(* IEC 61131-3 sources: MotionTestBenchMaster/Logical/00_AID/Libraries/Sidel_Libraries/SidelLog, 6 files *)

(* ---- SidelLog.typ ---- *)
(********************************************************************
 * COPYRIGHT --
 ********************************************************************
 * Library: SidelLog
 * File: SidelLog.typ
 * Author: Administrator
 * Created: July 15, 2014
 ********************************************************************
 * Data types of library SidelLog
 ********************************************************************)
(********************************                                    UPS LOG                                    **************************************************************)

TYPE
	Sidel_UpsIo_typ : 	STRUCT
		batteryAlarm : BOOL; (*True when the battery is failed*)
		batteryLow : BOOL; (*True when the battery is low*)
		shutdownReq : BOOL; (*Shutdown request*)
		noPowerSupply : BOOL; (*True when there is power supply*)
		shutdownAlarm : BOOL; (*True when the shutdown time exceed limits*)
		powerOffTime : UINT; (*Power off time*)
	END_STRUCT;
END_TYPE

(********************************                             SOFTWARE OBJECT LOG                **************************************************************)

TYPE
	MO_List_Light_typ : 	STRUCT
		name : ARRAY[0..13]OF SINT;
		grp : USINT;
		type : USINT;
		state : USINT;
		reserve : USINT;
		memtype : UDINT;
	END_STRUCT;
	SW_Obj_List : 	STRUCT
		version : MoVerStruc_typ; (*Version*)
		module : MO_List_Light_typ; (*Module details*)
	END_STRUCT;
END_TYPE

(* ---- LogSupplyEvents.st ---- *)
(********************************************************************
 * COPYRIGHT -- Bernecker + Rainer
 ********************************************************************
 * Library: GenUps
 * File: LogSupplyEvents.st
 * Author: gibertinim
 * Created: March 13, 2014
 ********************************************************************
 * Implementation of library GenUps
 ********************************************************************)

(* Write the power supply events in the specified logger *)
FUNCTION_BLOCK LogSupplyEvents

	IF (enable = TRUE) THEN

		CASE step OF

			0:
				pUpsIO ACCESS (ADR_UpsIO);

				errorID 			:=	ERR_FUB_BUSY;
				busy				:=	TRUE;
				error				:=	FALSE;
				noSupply			:= TRUE;
				batteryLow			:= FALSE;
				batteryAlarm		:= FALSE;
				shutdownRequested	:= FALSE;

				IF (customLogEntry_0.errorID = ERR_FUB_ENABLE_FALSE) THEN
					(* The function block started running *)
					step := 1;
				END_IF;

			1:

				memset(ADR(data),0,SIZEOF(data));
				customLogEntry_0.adrCustomEntry	:=	ADR(data);
				memset(ADR(tempString),0,SIZEOF(tempString));
				memset(ADR(tempString2),0,SIZEOF(tempString2));

				IF (pUpsIO.shutdownAlarm = TRUE) THEN
					step := 50;
				ELSE
					step := 51;
				END_IF;

			2:
				(* Waiting for an event *)

				IF 		((pUpsIO.batteryAlarm	= TRUE)		AND	(batteryAlarm		= FALSE))	THEN
					step := 10;
				ELSIF	((pUpsIO.batteryAlarm	= FALSE)	AND	(batteryAlarm		= TRUE))	THEN
					step := 11;
				ELSIF	((pUpsIO.batteryLow		= TRUE)		AND	(batteryLow			= FALSE))	THEN
					step := 20;
				ELSIF	((pUpsIO.batteryLow		= FALSE)	AND	(batteryLow			= TRUE))	THEN
					step := 21;
				ELSIF	((pUpsIO.noPowerSupply	= TRUE)		AND (noSupply			= FALSE))	THEN
					step := 30;
				ELSIF	((pUpsIO.noPowerSupply	= FALSE)	AND (noSupply			= TRUE))	THEN
					step := 31;
				ELSIF (pUpsIO.shutdownReq		= TRUE)		AND	(shutdownRequested	= FALSE)	THEN
					step := 40;
				ELSIF(	(pUpsIO.batteryAlarm	= FALSE)	AND	(batteryAlarm		= FALSE)	AND
						(pUpsIO.batteryLow		= FALSE)	AND	(batteryLow			= FALSE)	AND
						(pUpsIO.noPowerSupply	= FALSE)	AND (noSupply			= FALSE)	AND
						(pUpsIO.shutdownReq 	= FALSE)	AND (shutdownRequested	= FALSE))	THEN
					upsStatus := ERR_OK;
				ELSIF (	(pUpsIO.shutdownReq 	= FALSE)	AND (shutdownRequested	= TRUE)) THEN
					shutdownRequested := FALSE;
				END_IF;

			10:

				customLogEntry_0.enable 		:= 	TRUE;

				data.errorNum		:= ERR_UPS_BATTERY_FAULT;
				data.adr_string		:= ADR('UPS BATTERY FAULT');
				data.logLevel		:= arEVENTLOG_SEVERITY_WARNING;
				batteryAlarm		:= TRUE;
				upsStatus			:= ERR_UPS_BATTERY_FAULT;
				(* Waiting until the log is written succesfully *)
				IF (customLogEntry_0.errorID = ERR_OK) THEN
					(* Log entry written succesfully*)
					step 					:= 101;
					customLogEntry_0.enable := 	FALSE;
				ELSIF ((customLogEntry_0.errorID <> ERR_FUB_BUSY) AND (customLogEntry_0.errorID <> ERR_OK)AND (customLogEntry_0.errorID <> ERR_FUB_ENABLE_FALSE)) THEN
					(* Error occured while saving the logger *)
					errorStep	:= 10;
					errorID		:= customLogEntry_0.errorID;
					error		:= TRUE;
					step		:= 200;
				END_IF;

			11:
				(* Battery alarm recovered *)

				customLogEntry_0.enable := 	TRUE;
				data.errorNum			:= ERR_UPS_BATTERY_OK;

				data.adr_string	:= ADR('UPS BATTERY FAULT RECOVERED');
				data.logLevel	:= arEVENTLOG_SEVERITY_INFO;
				batteryAlarm	:= FALSE;
				(* Waiting until the log is written succesfully *)

				IF (customLogEntry_0.errorID = ERR_OK) THEN
					(* Log entry written succesfully*)
					step 					:= 101;
					customLogEntry_0.enable := FALSE;
				ELSIF ((customLogEntry_0.errorID <> ERR_FUB_BUSY) AND customLogEntry_0.errorID <> ERR_OK)AND (customLogEntry_0.errorID <> ERR_FUB_ENABLE_FALSE) THEN
					(* Error occured while saving the logger *)
					errorStep	:= 11;
					errorID		:= customLogEntry_0.errorID;
					error		:= TRUE;
					step		:= 200;
				END_IF;

			20:

				(* Battery low *)

				customLogEntry_0.enable 		:= 	TRUE;
				data.errorNum		:= ERR_UPS_BATTERY_LOW;
				data.adr_string		:= ADR('UPS BATTERY LOW');
				data.logLevel		:= arEVENTLOG_SEVERITY_WARNING;
				batteryLow			:= TRUE;
				upsStatus			:= ERR_UPS_BATTERY_LOW;
				(* Waiting until the log is written succesfully *)
				IF (customLogEntry_0.errorID = ERR_OK) THEN
					(* Log entry written succesfully*)
					step 					:= 101;
					customLogEntry_0.enable := FALSE;
				ELSIF ((customLogEntry_0.errorID <> ERR_FUB_BUSY) AND (customLogEntry_0.errorID <> ERR_OK)AND (customLogEntry_0.errorID <> ERR_FUB_ENABLE_FALSE)) THEN
					(* Error occured while saving the logger *)
					errorStep	:= 20;
					errorID		:= customLogEntry_0.errorID;
					error		:= TRUE;
					step		:= 200;
				END_IF;

			21:
				(* Battery recharged *)

				customLogEntry_0.enable 		:= 	TRUE;

				data.errorNum		:= ERR_UPS_BATTERY_CHARGED;
				data.adr_string		:= ADR('UPS BATTERY CHARGED');
				data.logLevel		:= arEVENTLOG_SEVERITY_INFO;
				batteryLow			:= FALSE;
				(* Waiting until the log is written succesfully *)

				IF (customLogEntry_0.errorID = ERR_OK) THEN
					(* Log entry written succesfully*)
					step 					:= 2;
					customLogEntry_0.enable := FALSE;
				ELSIF ((customLogEntry_0.errorID <> ERR_FUB_BUSY) AND (customLogEntry_0.errorID <> ERR_OK)AND (customLogEntry_0.errorID <> ERR_FUB_ENABLE_FALSE)) THEN
					(* Error occured while saving the logger *)
					errorStep	:= 21;
					errorID		:= customLogEntry_0.errorID;
					error		:= TRUE;
					step		:= 200;
				END_IF;

			30:

				(* Lost Power supply *)

				data.errorNum			:= ERR_UPS_NO_SUPPLY;
				data.adr_string			:= ADR('UPS NO POWER SUPPLY');
				data.logLevel			:= arEVENTLOG_SEVERITY_WARNING;
				noSupply				:= TRUE;
				upsStatus				:= ERR_UPS_NO_SUPPLY;
				customLogEntry_0.enable := 	TRUE;
				(* Waiting until the log is written succesfully *)
				IF (customLogEntry_0.errorID = ERR_OK) THEN
					(* Log entry written succesfully*)
					step 					:= 101;
					customLogEntry_0.enable := FALSE;
				ELSIF ((customLogEntry_0.errorID<> ERR_FUB_BUSY) AND (customLogEntry_0.errorID <> ERR_OK)AND (customLogEntry_0.errorID <> ERR_FUB_ENABLE_FALSE)) THEN
					(* Error occured while saving the logger *)
					errorStep	:= 30;
					errorID		:= customLogEntry_0.errorID;
					error		:= TRUE;
					step		:= 200;
				END_IF;

			31:
				(* Power supply ok *)

				customLogEntry_0.enable 		:= 	TRUE;

				data.errorNum		:= ERR_UPS_SUPPLY_BACK;
				data.adr_string		:= ADR('UPS POWER SUPPLY OK');
				data.logLevel		:= arEVENTLOG_SEVERITY_INFO;
				noSupply			:= FALSE;
				(* Waiting until the log is written succesfully *)
				IF (customLogEntry_0.errorID = ERR_OK) THEN
					(* Log entry written succesfully*)
					step 					:= 101;
					customLogEntry_0.enable := FALSE;
				ELSIF ((customLogEntry_0.errorID <> ERR_FUB_BUSY) AND (customLogEntry_0.errorID <> ERR_OK) AND (customLogEntry_0.errorID <> ERR_FUB_ENABLE_FALSE)) THEN
					(* Error occured while saving the logger *)
					errorStep	:= 31;
					errorID		:= customLogEntry_0.errorID;
					error		:= TRUE;
					step		:= 200;
				END_IF;

			40:
				(* Shutdown request *)

				customLogEntry_0.enable 		:= 	TRUE;

				data.errorNum		:= ERR_UPS_SHUTDOWN_REQ;
				data.adr_string		:= ADR('UPS SHUTDOWN REQUEST');
				data.logLevel		:= arEVENTLOG_SEVERITY_INFO;
				shutdownRequested	:= TRUE;
				upsStatus			:= ERR_UPS_SHUTDOWN_REQ;
				(* Waiting until the log is written succesfully *)
				IF (customLogEntry_0.errorID = ERR_OK) THEN
					(* Log entry written succesfully*)
					step 					:= 101;
					customLogEntry_0.enable := FALSE;
				ELSIF ((customLogEntry_0.errorID <> ERR_FUB_BUSY) AND (customLogEntry_0.errorID <> ERR_OK) AND (customLogEntry_0.errorID <> ERR_FUB_ENABLE_FALSE)) THEN
					(* Error occured while saving the logger *)
					errorStep	:= 40;
					errorID		:= customLogEntry_0.errorID;
					error		:= TRUE;
					step		:= 200;
				END_IF;

			50:
				(* Writing the total power off time to the logger *)
				(* Shutdown request *)
				itoa(pUpsIO.powerOffTime, ADR(tempString));
				tempString2 := 'UPS SHUTDOWN TIME ';
				strcat(ADR(tempString2), ADR(tempString));
				strcat(ADR(tempString2), ADR('s'));

				customLogEntry_0.enable 		:= 	TRUE;
				data.errorNum					:= ERR_UPS_SHUTDOWN_TIME;
				data.adr_string					:= ADR(tempString2);
				data.logLevel					:= arEVENTLOG_SEVERITY_INFO;
				shutdownRequested				:= TRUE;
				upsStatus						:= ERR_UPS_SHUTDOWN_REQ;

				(* Waiting until the log is written succesfully *)
				IF (customLogEntry_0.errorID = ERR_OK) THEN
					(* Log entry written succesfully*)
					step 					:= 51;
					customLogEntry_0.enable := FALSE;
				ELSIF ((customLogEntry_0.errorID <> ERR_FUB_BUSY) AND (customLogEntry_0.errorID <> ERR_OK) AND (customLogEntry_0.errorID <> ERR_FUB_ENABLE_FALSE)) THEN
					(* Error occured while saving the logger *)
					errorStep	:= 50;
					errorID		:= customLogEntry_0.errorID;
					error		:= TRUE;
					step		:= 200;
				END_IF;

			51:

				(* Identifier obtained succesfully *)
				IF (pUpsIO.noPowerSupply = TRUE) THEN
					step := 30;
				ELSE
					step := 31;
				END_IF;

			100:
				(* Waiting until the log is written succesfully *)
				IF (customLogEntry_0.errorID = ERR_OK) THEN
					(* Log entry written succesfully*)
					step := 101;

				ELSIF ((customLogEntry_0.errorID <> ERR_FUB_BUSY) AND (customLogEntry_0.errorID <> ERR_OK) AND (customLogEntry_0.errorID <> ERR_FUB_ENABLE_FALSE)) THEN
					(* Error occured while saving the logger *)
					errorStep	:= 100;
					errorID		:= customLogEntry_0.errorID;
					error		:= TRUE;
					step		:= 200;
				END_IF

			101:
			(* Disabling the function block *)
				IF (customLogEntry_0.errorID = ERR_FUB_ENABLE_FALSE) THEN
					memset(ADR(data),0,SIZEOF(data));
					step 			:= 2;
				END_IF;

			200:
			(* Error step *)
				customLogEntry_0.enable	:=	FALSE;

		END_CASE;

	ELSE

		error					:= TRUE;
		errorID					:= ERR_FUB_ENABLE_FALSE;
		customLogEntry_0.enable	:=	FALSE;
		step					:= 0;
		errorStep				:= 0;
		upsStatus				:= ERR_OK;
		noSupply				:= TRUE;
		batteryLow				:= FALSE;
		batteryAlarm			:= FALSE;
		shutdownRequested		:= FALSE;
		busy					:= FALSE;
		memset(ADR(data),0,SIZEOF(data));
	END_IF;

	customLogEntry_0();
END_FUNCTION_BLOCK

(* ---- SidelLog.fun ---- *)
(********************************************************************
 * COPYRIGHT --
 ********************************************************************
 * Library: SidelLog
 * File: SidelLog.fun
 * Author: Administrator
 * Created: July 15, 2014
 ********************************************************************
 * Functions and function blocks of library SidelLog
 ********************************************************************)

FUNCTION_BLOCK LogSupplyEvents (*Write the power supply events in the specified logger*)
	VAR_INPUT
		enable : BOOL; (*Enable the execution of the function block*)
		ADR_UpsIO : UDINT; (*Address of the UPS IO interface*)
	END_VAR
	VAR_OUTPUT
		errorID : DINT; (*Current error ID*)
		error : BOOL; (*True when the function block is in error*)
		upsStatus : UINT; (*Ups output status*)
		busy : BOOL; (*True when the function block is running*)
		errorStep : USINT; (*Error step*)
	END_VAR
	VAR
		step : USINT; (*Internal step*)
		batteryAlarm : BOOL; (*True when the battery is in alarm*)
		batteryLow : BOOL; (*True when the battery is low*)
		shutdownRequested : BOOL; (*Shutdown requested*)
		noSupply : BOOL; (*True wjen the power supply failed*)
		pUpsIO : REFERENCE TO Sidel_UpsIo_typ; (*Pointer to the UPS IO interface*)
		customLogEntry_0 : CustomLogEntry; (*Wrinting and getting information into a specified Logger*)
		tempString2 : STRING[80];
		tempString : STRING[80];
		data : pwr_log_custom_entry; (*Internal data to write*)
	END_VAR
END_FUNCTION_BLOCK

FUNCTION_BLOCK SynchLog (*Machine synchronization logger*)
	VAR_INPUT
		enable : BOOL; (*Enable the execution of the function block*)
		RAX1 : USINT;
		AXN : USINT;
		offsetAcquire : BOOL;
		testBit : USINT;
		axisNameHoming : STRING[80];
		axisName : STRING[80];
		positionMm : REAL;
		positionMmHoming : REAL;
	END_VAR
	VAR_OUTPUT
		errorID : DINT; (*Current error ID*)
		error : BOOL; (*True when the function block is in error*)
		testIndex : USINT;
		busy : BOOL; (*True when the function block is running*)
	END_VAR
	VAR
		step : USINT; (*Internal step*)
		errorStep : USINT; (*Error step*)
		indexAxis : USINT;
		phasingString : STRING[80];
		phasingAxisPosition : STRING[80];
		data : pwr_log_custom_entry; (*Wrinting and getting information into a specified Logger*)
		customLogEntry_0 : CustomLogEntry; (*Internal data to write*)
		rTrig_0 : R_TRIG;
	END_VAR
END_FUNCTION_BLOCK

FUNCTION_BLOCK SwChg (*Monitor and write into the user logger the canges of the software objects*)
	VAR_INPUT
		enable : BOOL; (*Enable the function block*)
		logLevel : USINT; (*Level of the log entry*)
		refreshTime : TIME; (*Refresh time*)
	END_VAR
	VAR_OUTPUT
		scan : BOOL; (*True when the module is getting the software object list*)
		searching : BOOL; (*True when the function block is searching for software object changes*)
		writingLog : BOOL; (*True when the funciton block is writing the entry into the logger*)
		waiting : BOOL; (*Waiting to search again*)
		busy : BOOL; (*True when the function block is busy*)
		error : BOOL; (*True when the function block is in error*)
		errorID : DINT; (*Actual error ID*)
	END_VAR
	VAR
		errorSubStep : USINT; (*Internal error SubStep*)
		errorStep : USINT; (*Internal erro Step*)
		step : USINT; (*Internal step*)
		substep : USINT; (*Internal substep*)
		cnt : UDINT; (*Internal counter*)
		mo_prev_index : UINT; (*List previous index*)
		mo_index : UINT; (*Actual index*)
		refresh : TON; (*Refresh timer*)
		waitWrite : TON; (*CF data object write delay*)
		customEntry : pwr_log_custom_entry; (*Custom log entry*)
		tempString : STRING[80]; (*Temporary string*)
		tempModule : MO_List_typ; (*Temporary module informations*)
		nrChanges : UINT; (*Number of changed elements*)
		swListTempID : UDINT; (*Temporary software list ID*)
		swListID : UDINT; (*Software list ID*)
		iOldList : ARRAY[0..iMaxEntries] OF SW_Obj_List; (*Internal Old List*)
		iActList : ARRAY[0..iMaxEntries] OF SW_Obj_List; (*Internal Actual List*)
	END_VAR
	VAR CONSTANT
		CST_fwOBJ : USINT := 132; (*Firmware Object*)
		CST_configOBJ : USINT := 67; (*Configuration Object*)
		CST_hwOBJ : USINT := 43; (*Hrdwa object*)
		CST_ncOBJ : USINT := 70; (*NC Object*)
		CST_cycOBJ : USINT := 17; (*Cyclic Object*)
		CST_sysOBJ : USINT := 18; (*System Object*)
		iMaxEntries : UINT := 999; (*Internal number of entries*)
	END_VAR
	VAR
		writeDiff : CustomLogEntry; (*Writes the custom information into the logger*)
		datObjWrite_0 : DatObjWrite; (*Write into a data Object*)
		datObjRead_0 : DatObjRead; (*Read data from a data Object*)
		datObjInfo_0 : DatObjInfo; (*Get the informations from a data object*)
		datObjCopy_0 : DatObjCopy; (*Copy a data object*)
		datObjCreate_0 : DatObjCreate; (*Create a data object*)
		datObjDelete_0 : DatObjDelete; (*Delete a data object*)
		actListElements : UINT; (*Number of entries in the actual list*)
		oldListElements : UINT; (*Number of entries in the old list*)
		newSwListT : BOOL; (*Software list data object present*)
		oldSubStep : USINT;
	END_VAR
END_FUNCTION_BLOCK

(* ---- SwChg.st ---- *)
(********************************************************************
 * COPYRIGHT --
 ********************************************************************
 * Library: Powertoys
 * File: swChg.st
 * Author: Massimo Gibertini
 * Created: August 07, 2014
 ********************************************************************
 * Implementation of library Powertoys
 ********************************************************************)

(* Monitor and write into the user logger the canges of the software objects *)
FUNCTION_BLOCK SwChg

	IF (enable = TRUE) THEN
		customEntry.logLevel 		:= logLevel;
		waitWrite.PT				:= T#10m;

		CASE step OF

			0:
				(* Getting the software list *)
				busy			:= TRUE;
				searching		:= FALSE;
				writingLog		:= FALSE;
				waiting			:= FALSE;
				scan			:= TRUE;
				error			:= FALSE;
				errorID			:= ERR_FUB_BUSY;

				CASE substep OF

					0:
						memset(ADR(tempModule),0,SIZEOF(tempModule));
						memset(ADR(iActList),0,SIZEOF(iActList));
						memset(ADR(iOldList),0,SIZEOF(iOldList));

						(* Checking if the swList temporary data object exist in the userRam or not*)
						datObjInfo_0.pName 	:= ADR(swListTempDataObjName);
						datObjInfo_0.enable	:= TRUE;
						substep 			:= 1;

					1:
						datObjInfo_0();
						IF (datObjInfo_0.status = doERR_MODULNOTFOUND) THEN
							(* Temporary data object not found *)
							swListTempID	:= 0;
							substep			:= 5;
						ELSIF (datObjInfo_0.status = ERR_OK) THEN
							(* Data object found *)
							swListTempID	:= datObjInfo_0.ident;
							//substep			:= 2;
							substep			:= 5;
						ELSIF (datObjInfo_0.status <> ERR_OK) AND (datObjInfo_0.status <> doERR_MODULNOTFOUND) AND (datObjInfo_0.status <> ERR_FUB_BUSY) THEN
							errorID			:= datObjInfo_0.status;
							errorStep		:= step;
							errorSubStep	:= substep;
							step 			:= 200;
							substep			:= 0;
						END_IF;

					2:
						datObjInfo_0.enable	:= FALSE;
						datObjInfo_0();
						IF (datObjInfo_0.status = ERR_FUB_ENABLE_FALSE) THEN
							substep			:= 3;
						END_IF;

					3:
						(* Delete the temporary data object *)
						datObjDelete_0.ident	:= swListTempID;
						datObjDelete_0.enable	:= TRUE;
						substep					:= 4;

					4:
						datObjDelete_0();
						IF (datObjDelete_0.status = ERR_OK) THEN
							substep			:= 5;
							swListTempID	:= 0;
						ELSIF (datObjDelete_0.status <> ERR_OK) AND (datObjDelete_0.status <> ERR_FUB_BUSY) THEN
							errorID			:= datObjDelete_0.status;
							errorStep		:= step;
							errorSubStep	:= substep;
							step 			:= 200;
							substep			:= 0;
						END_IF;

					5:
						(* Disable fub *)
						datObjDelete_0.enable	:= FALSE;
						datObjDelete_0();
						datObjInfo_0.enable	:= FALSE;
						datObjInfo_0();
						IF (datObjDelete_0.status = ERR_FUB_ENABLE_FALSE) AND (datObjInfo_0.status = ERR_FUB_ENABLE_FALSE) THEN
							substep				:= 6;
						END_IF;

					6:
						(* temporary data object not present or deleted *)
						(* Checking if the swList data object exist or not *)
						datObjInfo_0.pName 	:= ADR(swListDatObjName);
						datObjInfo_0.enable	:= TRUE;
						datObjInfo_0();
						IF (datObjInfo_0.status <> ERR_FUB_BUSY) AND (datObjInfo_0.status <> ERR_FUB_ENABLE_FALSE) THEN
							substep := 7;
						END_IF;

					7:
						datObjInfo_0();
						IF (datObjInfo_0.status = doERR_MODULNOTFOUND) THEN
							(* Data object not found *)
							swListID		:= 0;
							substep			:= 100;
						ELSIF (datObjInfo_0.status = doERR_CHECKSUM_WARNING) THEN
							swListID		:= datObjInfo_0.ident;
							substep			:= 10;
						ELSIF (datObjInfo_0.status = ERR_OK) THEN
							(* Data object found *)
							swListID		:= datObjInfo_0.ident;
							IF (swListTempID = 0) THEN
								substep			:= 50;
							ELSE
								substep 		:= 150;
							END_IF;

						ELSIF (datObjInfo_0.status <> ERR_OK) AND (datObjInfo_0.status <> doERR_CHECKSUM_WARNING) AND (datObjInfo_0.status <> doERR_MODULNOTFOUND) AND (datObjInfo_0.status <> ERR_FUB_BUSY) THEN
							errorID			:= datObjInfo_0.status;
							errorStep		:= step;
							errorSubStep	:= substep;
							step 			:= 200;
							substep			:= 0;
						END_IF;

					(* Data object damaged, deleting *)
					10:
						datObjInfo_0.enable	:= FALSE;
						datObjInfo_0();
						IF (datObjInfo_0.status = ERR_FUB_ENABLE_FALSE) THEN
							substep			:= 11;
						END_IF;

					11:
						datObjDelete_0.ident	:= swListID;
						datObjDelete_0.enable	:= TRUE;
						datObjDelete_0();
						IF (datObjDelete_0.status <> ERR_FUB_BUSY) AND (datObjDelete_0.status <> ERR_FUB_ENABLE_FALSE) THEN
							substep 				:= 12;
						END_IF;

					12:
						datObjDelete_0();
						IF (datObjDelete_0.status = ERR_OK) THEN
							substep				:= 13;
						ELSIF (datObjDelete_0.status <> ERR_OK) AND (datObjDelete_0.status <> ERR_FUB_BUSY) THEN
							errorID				:= datObjDelete_0.status;
							errorStep			:= step;
							errorSubStep		:= substep;
							step 				:= 200;
							substep				:= 0;
						END_IF;

					13:
						datObjDelete_0.enable	:= FALSE;
						datObjDelete_0();
						IF (datObjDelete_0.status = ERR_FUB_ENABLE_FALSE) THEN
							(* No existing data object *)
							substep 			:= 100;
							swListID 			:= 0;
						END_IF;

					50:
						(* swList data object present, copy to DRam *)
						datObjInfo_0.enable			:= FALSE;
						datObjCopy_0.ident 			:= swListID;
						datObjCopy_0.pNameTarget 	:= ADR(swListTempDataObjName);
						datObjCopy_0.MemTypeTarget	:= doTEMP;
						datObjCopy_0.enable			:= TRUE;
						datObjCopy_0();
						substep := 51;

					51:
						datObjCopy_0();
						IF (datObjCopy_0.status = ERR_OK) THEN
							substep 				:= 52;
							swListTempID			:= datObjCopy_0.identNew;
						ELSIF (datObjCopy_0.status <> ERR_OK) AND (datObjCopy_0.status <> ERR_FUB_BUSY) THEN
							errorID					:= datObjCopy_0.status;
							errorStep				:= step;
							errorSubStep			:= substep;
							step 					:= 200;
							substep					:= 0;
						END_IF;

					52:
						datObjCopy_0.enable			:= FALSE;
						datObjCopy_0();
						IF (datObjCopy_0.status = ERR_FUB_ENABLE_FALSE) THEN
							(* Temporary Data object recovered succesfully *)
							substep					:= 150;

						END_IF;

					100:
						(* Creating the temporary data object*)
						IF (swListTempID = 0) THEN
							datObjInfo_0.enable		:= FALSE;
							datObjCreate_0.grp		:= 0;
							datObjCreate_0.pName	:= ADR(swListTempDataObjName);
							datObjCreate_0.len		:= SIZEOF(iActList);
							datObjCreate_0.MemType	:= doTEMP;
							datObjCreate_0.Option	:= doNO_CS;
							datObjCreate_0.pCpyData	:= ADR(iActList);
							datObjCreate_0.enable	:= TRUE;
							datObjCreate_0();
							substep					:= 101;
						ELSE
							substep					:= 110;
						END_IF;

					101:
						datObjCreate_0();
						IF (datObjCreate_0.status = ERR_OK) THEN
							substep				:= 102;
							swListTempID		:= datObjCreate_0.ident;
							newSwListT			:= TRUE;
						ELSIF (datObjCreate_0.status <> ERR_OK) AND (datObjCreate_0.status <> ERR_FUB_BUSY) THEN
							errorID				:= datObjCreate_0.status;
							errorStep			:= step;
							errorSubStep		:= substep;
							step 				:= 200;
							substep				:= 0;
						END_IF;

					102:
						datObjCreate_0.enable	:= FALSE;
						datObjCreate_0();
						IF (datObjCreate_0.status = ERR_FUB_ENABLE_FALSE) THEN
							substep				:= 110;

						END_IF;

					110:
						(* Creating the cf data object*)
						datObjCreate_0.grp		:= 0;
						datObjCreate_0.pName	:= ADR(swListDatObjName);
						datObjCreate_0.len		:= SIZEOF(iOldList);
						datObjCreate_0.MemType	:= doUSRROM;
						datObjCreate_0.Option	:= 0;
						datObjCreate_0.pCpyData	:= ADR(iOldList);
						datObjCreate_0.enable	:= TRUE;
						substep					:= 112;

					112:
						datObjCreate_0();
						IF (datObjCreate_0.status = ERR_OK) THEN
							substep					:= 113;
							swListID				:= datObjCreate_0.ident;
							datObjCreate_0.enable	:= FALSE;
						ELSIF (datObjCreate_0.status <> ERR_OK) AND (datObjCreate_0.status <> ERR_FUB_BUSY) THEN
							errorID					:= datObjCreate_0.status;
							errorStep				:= step;
							errorSubStep			:= substep;
							step 					:= 200;
							substep					:= 0;
						END_IF;

					113:
						datObjCreate_0.enable		:= FALSE;
						datObjCreate_0();
						IF (datObjCreate_0.status = ERR_FUB_ENABLE_FALSE) AND newSwListT THEN
							substep					:= 200;
							oldListElements			:= 0;
						ELSIF (datObjCreate_0.status = ERR_FUB_ENABLE_FALSE) AND NOT (newSwListT) THEN
							substep					:= 150;
							oldListElements			:= 0;
						END_IF;

					150:
						(* Loading the existing temporary data object *)
						datObjRead_0.ident			:= swListTempID;
						datObjRead_0.Offset			:= 0;
						datObjRead_0.pDestination	:= ADR(iOldList);
						datObjRead_0.len			:= SIZEOF(iOldList);
						datObjRead_0.enable			:= TRUE;
						datObjRead_0();
						substep						:= 151;

					151:

						datObjRead_0();
						IF (datObjRead_0.status = ERR_OK) THEN
							substep					:= 152;
						ELSIF (datObjRead_0.status <> ERR_OK) AND (datObjRead_0.status <> ERR_FUB_BUSY)	THEN
							errorID					:= datObjRead_0.status;
							errorStep				:= step;
							errorSubStep			:= substep;
							step 					:= 200;
							substep					:= 0;
						END_IF;

					152:
						datObjRead_0.enable			:= FALSE;
						datObjRead_0();
						IF (datObjRead_0.status = ERR_FUB_ENABLE_FALSE) THEN
							oldListElements 		:= 0;
							substep 				:= 153;
						END_IF;

					153:
						(* Listing the number of entries in the old list *)
						memset(ADR(tempString),0,SIZEOF(tempString));
						memcpy(ADR(tempString),ADR(iOldList[oldListElements].module.name[0]),SIZEOF(iOldList[oldListElements].module.name));
						IF (tempString <> '') THEN
							oldListElements := oldListElements + 1;
						ELSE
							substep 		:= 200;
						END_IF;

					200:
						(* Cleaning the memory of the actual list *)
						(* Listing all the software objects *)
						memset(ADR(iActList),0,SIZEOF(iActList));
						mo_prev_index 	:= 16#FFFF;
						mo_index 		:= 0;
						nrChanges 		:= 0;
						substep			:= 201;

					201:
						(* Listing all the software objects element *)
						memset(ADR(tempModule), 0, SIZEOF(tempModule));
						MO_list(mo_prev_index, ADR(mo_index),ADR(tempModule));

						IF (tempModule.type <> 0) AND ((tempModule.type = CST_configOBJ)	OR
							(tempModule.type = CST_cycOBJ)		OR
							(tempModule.type = CST_fwOBJ)		OR
							(tempModule.type = CST_hwOBJ)		OR
							(tempModule.type = CST_ncOBJ)		OR
							(tempModule.type = CST_sysOBJ))		THEN

							(* Valid system object *)
							MO_ver(ADR(tempModule.name),0,ADR(iActList[nrChanges].version));
							memcpy(ADR(iActList[nrChanges].module.name[0]),ADR(tempModule.name[0]), SIZEOF(tempModule.name));

							iActList[nrChanges].module.grp		:= tempModule.grp;
							iActList[nrChanges].module.memtype	:= tempModule.memtype;
							iActList[nrChanges].module.reserve 	:= tempModule.reserve;
							iActList[nrChanges].module.state	:= tempModule.state;
							iActList[nrChanges].module.type		:= tempModule.type;

							nrChanges							:= nrChanges + 1;
							substep 							:= 202;
						ELSE
							substep 							:= 202;
						END_IF;

					202:
						(* Checking if I have finished to scan *)

						IF (mo_prev_index = mo_index) OR (nrChanges = iMaxEntries) THEN
							substep 		:= 203;
						ELSE
							mo_prev_index	:= mo_index;
							substep 		:= 201;
						END_IF;

					203:
						(* Software list complete *)
						actListElements 	:= nrChanges;
						step 				:= 1;
						substep 			:= 0;

				END_CASE;

			1:
				(* Searching for modified software objects *)
				busy			:= TRUE;
				searching		:= TRUE;
				writingLog		:= FALSE;
				waiting			:= FALSE;
				scan			:= FALSE;
				error			:= FALSE;
				errorID			:= ERR_FUB_BUSY;

				CASE substep OF
					0:
						(* Software list complete, comparing memory area *)
						IF (memcmp(ADR(iActList), ADR(iOldList), SIZEOF(iActList)) = 0) THEN

							(* No software changes *)
							substep	:= 0;
							step	:= 20;

						ELSE

							(* There are some changes *)
							substep		:= 1;
							cnt			:= 0;
							nrChanges	:= 0;
							oldSubStep	:= 0;
						END_IF;

					1:
						(* Trying to find the module in the same position of the old array *)
						(* First speed up improvement *)
						IF ((memcmp(ADR(iActList[nrChanges].module.name[0]), ADR(iOldList[nrChanges].module.name[0]), SIZEOF(iOldList[nrChanges].module.name)) = 0)
							AND (cnt < oldListElements) AND (nrChanges < actListElements)) THEN

							(* Module found *)
							IF (memcmp(ADR(iActList[nrChanges]),ADR(iOldList[nrChanges]),SIZEOF(iOldList[nrChanges])) = 0) THEN

								(* The module are the same *)
								nrChanges	:= nrChanges + 1;
								cnt			:= 0;
							ELSE

								(* The module is modified *)
								substep 	:= 10;
								step		:= 10;

							END_IF;

						ELSE
							(* Module not found *)
							substep 	:= 10;

						END_IF;

					10:
						(* Comparing the all elements of the iActList with all the elements of iOldList to find if the element exist or not *)
						IF (memcmp(ADR(iActList[nrChanges].module.name[0]), ADR(iOldList[cnt].module.name[0]), SIZEOF(iOldList[cnt].module.name)) <> 0) AND (nrChanges < actListElements) THEN
							IF (cnt < oldListElements)  THEN
								(* Module not found *)
								cnt 		:= cnt + 1;

							ELSIF (cnt >= oldListElements)  THEN

								(* New software module *)
								substep		:= 20;
								step		:= 10;
							END_IF;

						ELSIF ((memcmp(ADR(iActList[nrChanges].module.name[0]), ADR(iOldList[cnt].module.name[0]), SIZEOF(iOldList[cnt].module.name)) = 0)
								AND (cnt < oldListElements) AND (nrChanges < actListElements)) THEN

							(* Module found *)
							IF (memcmp(ADR(iActList[nrChanges]),ADR(iOldList[cnt]),SIZEOF(iOldList[cnt])) = 0) THEN

								(* The module are the same *)
								nrChanges	:= nrChanges + 1;
								cnt			:= 0;
								substep 	:= 1;
							ELSE

								(* The module is modified *)
								substep 	:= 10;
								step		:= 10;
							END_IF;

						ELSIF (nrChanges >= actListElements) THEN

							(* Search finished, checking the removed objects *)
							substep			:= 2;
							cnt 			:= 0;
							nrChanges 		:= 0;
						END_IF;

					2:
						(* Trying to find the module in the same position of the old array *)
						(* Second speed up improvement *)
						IF ((memcmp(ADR(iActList[cnt].module.name[0]), ADR(iOldList[cnt].module.name[0]), SIZEOF(iOldList[cnt].module.name)) = 0)
							AND (cnt < oldListElements) AND (nrChanges < actListElements)) THEN

							(* Module found *)
							cnt				:= cnt + 1;
							nrChanges		:= 0;

						ELSE
							(* Module not found *)
							nrChanges		:= 0;
							substep 	:= 20;
						END_IF

					20:
						(* Checking if there are any removed software object *)
						IF (memcmp(ADR(iActList[nrChanges].module.name[0]), ADR(iOldList[cnt].module.name[0]), SIZEOF(iOldList[cnt].module.name)) <> 0) AND (oldListElements <> 0) AND (cnt < oldListElements) THEN

							IF  (nrChanges < actListElements) THEN

								(* Module not found *)
								nrChanges	:= nrChanges + 1;

							ELSIF (nrChanges >= actListElements) THEN

								(* SW module removed *)
								substep 	:= 0;
								step		:= 10;
							END_IF;

						ELSIF ((memcmp(ADR(iActList[nrChanges].module.name[0]), ADR(iOldList[cnt].module.name[0]), SIZEOF(iOldList[cnt].module.name)) = 0)
							AND (cnt < oldListElements) AND (nrChanges < actListElements)) THEN

							(* Module found *)
							cnt				:= cnt + 1;
							substep 		:= 2;
							nrChanges		:= 0;

						ELSIF (cnt >= oldListElements) THEN

							(* Search finished *)
							step			:= 10;
							substep 		:= 30;
							cnt				:= 0;
							nrChanges		:= 0;
						END_IF;

				END_CASE;

			10:
				(* Writing informations into the logger and data object *)
				busy 			:= TRUE;
				searching 		:= FALSE;
				writingLog		:= TRUE;
				waiting 		:= FALSE;
				scan			:= FALSE;
				error			:= FALSE;
				errorID			:= ERR_FUB_BUSY;

				CASE substep OF

					0:
						(* Removed software module *)
						memset(ADR(tempString),0,SIZEOF(tempString));
						tempString	:= 'REMOVED SW MODULE: ';
						memcpy(ADR(tempString)+LEN(tempString),ADR(iOldList[cnt].module.name[0]), SIZEOF(iOldList[cnt].module.name));
						substep		:= 1;

					1:
						(* Writing into the logger *)
						customEntry.adr_string 		:= ADR(tempString);
						customEntry.errorNum 		:= LOG_SW_OBJ_CHG;
						writeDiff.adrCustomEntry 	:= ADR(customEntry);
						writeDiff.enable 			:= TRUE;
						substep 					:= 2;

					2:

						IF (writeDiff.done = TRUE) THEN
							substep			:= 3;
						ELSIF (writeDiff.error) THEN
							errorID			:= writeDiff.errorID;
							errorStep		:= step;
							errorSubStep	:= substep;
							step 			:= 200;
							substep			:= 0;
						END_IF;

					3:
						writeDiff.enable	:= FALSE;
						IF (writeDiff.errorID = ERR_FUB_ENABLE_FALSE) THEN
							cnt				:= cnt + 1;
							nrChanges		:= 0;
							step			:= 1;
							substep			:= 2;
						END_IF;

					10:
						(* Modified software module *)
						memset(ADR(tempString),0,SIZEOF(tempString));
						tempString	:= 'MODIFIED SW MODULE: ';
						memcpy(ADR(tempString)+LEN(tempString),ADR(iActList[nrChanges].module.name[0]), SIZEOF(iActList[nrChanges].module.name));
						substep		:= 11;

					11:
						(* Writing into the logger *)
						customEntry.adr_string 		:= ADR(tempString);
						customEntry.errorNum 		:= LOG_SW_OBJ_CHG;
						writeDiff.adrCustomEntry 	:= ADR(customEntry);
						writeDiff.enable 			:= TRUE;
						substep 					:= 12;

					12:

						IF (writeDiff.done = TRUE) THEN
							substep			:= 13;
						ELSIF (writeDiff.error) THEN
							errorID			:= writeDiff.errorID;
							errorStep		:= step;
							errorSubStep	:= substep;
							step 			:= 200;
							substep			:= 0;
						END_IF;

					13:
						writeDiff.enable	:= FALSE;
						IF (writeDiff.errorID = ERR_FUB_ENABLE_FALSE) THEN
							cnt				:= 0;
							nrChanges		:= nrChanges + 1;
							substep			:= 1;
							step			:= 1;
						END_IF;

					20:
						(* New software module *)
						memset(ADR(tempString),0,SIZEOF(tempString));
						tempString	:= 'NEW SW MODULE: ';
						memcpy(ADR(tempString)+LEN(tempString),ADR(iActList[nrChanges].module.name[0]), SIZEOF(iActList[nrChanges].module.name));
						substep		:= 21;

					21:
						(* Writing into the logger *)
						customEntry.adr_string 		:= ADR(tempString);
						customEntry.errorNum 		:= LOG_SW_OBJ_NEW;
						writeDiff.adrCustomEntry 	:= ADR(customEntry);
						writeDiff.enable 			:= TRUE;
						substep						:= 22;

					22:
						IF (writeDiff.done = TRUE) THEN
							substep			:= 23;
						ELSIF (writeDiff.error) THEN
							errorID			:= writeDiff.errorID;
							errorStep		:= step;
							errorSubStep	:= substep;
							step 			:= 200;
							substep			:= 0;
						END_IF;

					23:
						writeDiff.enable	:= FALSE;
						IF (writeDiff.errorID = ERR_FUB_ENABLE_FALSE) THEN
							cnt				:= 0;
							nrChanges		:= nrChanges + 1;
							substep			:= 1;
							step			:= 1;
						END_IF;

					30:
						(* Writing temporary data object *)
						datObjWrite_0.ident		:= swListTempID;
						datObjWrite_0.len		:= SIZEOF(iActList);
						datObjWrite_0.Offset	:= 0;
						datObjWrite_0.pSource	:= ADR(iActList);
						datObjWrite_0.enable	:= TRUE;
						datObjWrite_0();
						substep					:= 31;

					31:
						datObjWrite_0();
						IF (datObjWrite_0.status = ERR_OK) THEN
							substep 				:= 50;
							waitWrite.IN 			:= TRUE;
							datObjWrite_0.enable 	:= FALSE;
						ELSIF (datObjWrite_0.status <> ERR_OK) AND (datObjWrite_0.status <> ERR_FUB_BUSY) THEN
							errorID					:= datObjWrite_0.status;
							errorStep				:= step;
							errorSubStep			:= substep;
							step 					:= 200;
							substep					:= 0;
						END_IF;

					40:
						(* Writing cf data object *)
						datObjWrite_0.ident			:= swListID;
						datObjWrite_0.len			:= SIZEOF(iActList);
						datObjWrite_0.Offset		:= 0;
						datObjWrite_0.pSource		:= ADR(iActList);
						datObjWrite_0.enable		:= TRUE;
						datObjWrite_0();
						substep						:= 41;
					41:
						datObjWrite_0();
						IF (datObjWrite_0.status = ERR_OK) THEN
							substep 				:= 50;
							waitWrite.IN 			:= FALSE;
							datObjWrite_0.enable 	:= FALSE;
						ELSIF (datObjWrite_0.status <> ERR_OK) AND (datObjWrite_0.status <> ERR_FUB_BUSY) THEN
							errorID					:= datObjWrite_0.status;
							errorStep				:= step;
							errorSubStep			:= substep;
							step 					:= 200;
							substep					:= 0;
						END_IF;

					50:
						(* Copy the actual list into the old list *)
						memcpy(ADR(iOldList), ADR(iActList), SIZEOF(iActList));
						memset(ADR(tempString),0,SIZEOF(tempString));
						substep := 0;
						step 	:= 20;
				END_CASE;

			20:
				(* Waiting step *)
				busy 			:= TRUE;
				searching 		:= FALSE;
				writingLog		:= FALSE;
				waiting 		:= TRUE;
				scan			:= FALSE;
				error			:= FALSE;
				errorID			:= ERR_FUB_BUSY;

				CASE substep OF
					0:
						(* No software changes *)
						refresh.PT := refreshTime;
						refresh.IN := TRUE;

						IF refresh.Q THEN
							substep := 1;
						END_IF;

					1:
						(* Refresh time elapsed *)
						IF (waitWrite.Q) THEN
							step 	:= 10;
							substep := 40;
						ELSE
							refresh.IN := FALSE;
							step 	:= 0;
							substep := 152;
						END_IF;

				END_CASE;

			200:
				(* Error state resetting all the used function block *)
				writeDiff.enable		:= FALSE;
				refresh.IN 				:= FALSE;
				waitWrite.IN			:= FALSE;
				datObjWrite_0.enable	:= FALSE;
				datObjInfo_0.enable		:= FALSE;
				datObjDelete_0.enable	:= FALSE;
				datObjRead_0.enable		:= FALSE;
				datObjCreate_0.enable	:= FALSE;
				datObjCopy_0.enable		:= FALSE;

				(* Updating the status *)
				busy			:= FALSE;
				searching		:= FALSE;
				writingLog		:= FALSE;
				waiting			:= FALSE;
				scan			:= FALSE;
				error			:= TRUE;
		END_CASE;

	ELSE

		mo_prev_index 	:= 16#FFFF;
		mo_index 		:= 0;
		cnt 			:= 0;
		nrChanges 		:= 0;
		substep			:= 0;
		step			:= 0;
		errorSubStep	:= 0;
		errorStep		:= 0;
		oldSubStep		:= 0;

		oldListElements := 0;
		actListElements	:= 0;

		error			:= TRUE;
		errorID			:= ERR_FUB_ENABLE_FALSE;
		busy			:= FALSE;
		searching		:= FALSE;
		writingLog		:= FALSE;
		waiting			:= FALSE;
		scan			:= FALSE;
		newSwListT		:= FALSE;
		(* Resetting all the used function block *)
		writeDiff.enable		:= FALSE;
		refresh.IN 				:= FALSE;
		waitWrite.IN			:= FALSE;
		datObjWrite_0.enable	:= FALSE;
		datObjInfo_0.enable		:= FALSE;
		datObjDelete_0.enable	:= FALSE;
		datObjRead_0.enable		:= FALSE;
		datObjCreate_0.enable	:= FALSE;
		datObjCopy_0.enable		:= FALSE;
	END_IF;

	writeDiff();
	refresh();
	waitWrite();

END_FUNCTION_BLOCK

(* ---- SynchLog.st ---- *)
(********************************************************************
 * COPYRIGHT --
 ********************************************************************
 * Library: SidelLog
 * File: SynchLog.st
 * Author: Administrator
 * Created: July 15, 2014
 ********************************************************************
 * Implementation of library SidelLog
 ********************************************************************)

(* Machine synchronization logger *)
FUNCTION_BLOCK SynchLog

	IF (enable = TRUE) THEN

		CASE step OF

			0:

				errorID 			:=	ERR_FUB_BUSY;
				busy				:=	TRUE;
				error				:=	FALSE;

				IF (customLogEntry_0.errorID = ERR_FUB_ENABLE_FALSE) THEN
					(* The function block started running *)
					step := 1;
				END_IF;

			1:
				memset(ADR(data),0,SIZEOF(data));

				data.adr_string			:= 	ADR(phasingString);

				customLogEntry_0.adrCustomEntry	:=	(ADR(data));

				rTrig_0.CLK				:=	offsetAcquire;
				customLogEntry_0.enable	:=	FALSE;

				IF rTrig_0.Q	=	TRUE THEN
					step					:=	2;
				END_IF;

			2:
				customLogEntry_0.enable	:=	TRUE;

				data.errorNum	:= LOG_SYNC_AXIS;
				data.logLevel	:= arEVENTLOG_SEVERITY_INFO;

				phasingString	:=	'Homing of Axis ';
				strcat(ADR(phasingString),ADR(axisNameHoming));
				strcat(ADR(phasingString), ADR(' DONE , old position '));
				ftoa(positionMmHoming,ADR(phasingAxisPosition));
				strcat(ADR(phasingString),ADR(phasingAxisPosition));
				strcat(ADR(phasingString), ADR('mm'));

				IF customLogEntry_0.errorID = ERR_OK THEN
					step					:=	10;
					customLogEntry_0.enable	:=	FALSE;
					indexAxis				:=	RAX1;

				ELSIF	((customLogEntry_0.errorID <> ERR_FUB_BUSY) AND (customLogEntry_0.errorID <> ERR_OK)AND (customLogEntry_0.errorID <> ERR_FUB_ENABLE_FALSE)) THEN
					errorStep	:= 	2;
					errorID		:=	customLogEntry_0.errorID;
					error		:=	TRUE;
					step		:=	200;
				END_IF;

			10:
				IF (customLogEntry_0.errorID=ERR_FUB_ENABLE_FALSE) THEN

					step		:=	20;
					indexAxis	:=	RAX1;
					testIndex	:=  RAX1;
				END_IF;

			20:
				IF indexAxis <= AXN THEN

					IF testBit = TRUE THEN

						customLogEntry_0.enable	:=	TRUE;
						data.errorNum	:= LOG_AXIS_POSITION;
						data.logLevel	:= arEVENTLOG_SEVERITY_INFO;

						phasingString	:=	'Position of Axis ';
						strcat(ADR(phasingString),ADR(axisName));
						strcat(ADR(phasingString), ADR(' is '));
						ftoa(positionMm,ADR(phasingAxisPosition));
						strcat(ADR(phasingString),ADR(phasingAxisPosition));
						strcat(ADR(phasingString), ADR('mm'));

						IF customLogEntry_0.errorID = ERR_OK THEN

							customLogEntry_0.enable	:=	FALSE;
							step					:=21;
						ELSIF	((customLogEntry_0.errorID <> ERR_FUB_BUSY) AND (customLogEntry_0.errorID <> ERR_OK)AND (customLogEntry_0.errorID <> ERR_FUB_ENABLE_FALSE)) THEN
							errorStep	:= 20;
							errorID		:= customLogEntry_0.errorID;
							error		:= TRUE;
							step		:=	200;

						END_IF;

					ELSE
						indexAxis	:=	indexAxis+1;
						testIndex	:=	indexAxis;
					END_IF;
				ELSE

					step	:=	1;

				END_IF;
			21:
				IF (customLogEntry_0.errorID=ERR_FUB_ENABLE_FALSE) THEN
					step		:=	20;
					indexAxis	:=	indexAxis+1;
					testIndex	:=	indexAxis;
				END_IF;

			200:
				customLogEntry_0.enable	:=	FALSE;

		END_CASE;

	ELSE

				error					:=	TRUE;
				errorID					:=	ERR_FUB_ENABLE_FALSE;
				customLogEntry_0.enable	:=	FALSE;
				step					:=	0;
				testIndex				:=	0;
				memset(ADR(data),0,SIZEOF(data));
	END_IF;

	customLogEntry_0();
	rTrig_0();

END_FUNCTION_BLOCK

(* ---- SidelLog.var ---- *)
(********************************************************************
 * COPYRIGHT --
 ********************************************************************
 * Library: SidelLog
 * File: SidelLog.var
 * Author: Administrator
 * Created: July 15, 2014
 ********************************************************************
 * Constants of library SidelLog
 ********************************************************************)
(*************************************************************************************                                UPS LOGGER                       ****************************************************************************************)
VAR CONSTANT
	ERR_UPS_BATTERY_FAULT : UINT := 55000; (*Ups battery fault*)
	ERR_UPS_BATTERY_OK : UINT := 55001; (*Ups battery ok*)
	ERR_UPS_BATTERY_CHARGED : UINT := 55002; (*Ups  battery charged*)
	ERR_UPS_BATTERY_LOW : UINT := 55003; (*Ups battery low*)
	ERR_UPS_SUPPLY_BACK : UINT := 55004; (*Returned back the power supply*)
	ERR_UPS_NO_SUPPLY : UINT := 55005; (*Ups no power spply*)
	ERR_UPS_SHUTDOWN_REQ : UINT := 55006; (*Ups shutdown request*)
	ERR_UPS_SHUTDOWN_TIME : UINT := 50007; (*Ups shutdown time*)
END_VAR
(************************************************************************************                 MACHINE SYNCHRONIZATION            ****************************************************************************************)
VAR CONSTANT
	LOG_AXIS_POSITION : UINT := 55010; (*Axis position during machine synchronization*)
	LOG_SYNC_AXIS : UINT := 55011; (*Synchronized axis*)
END_VAR
(************************************************************************************                 SOFTWARE OBJECT MONITOR           ****************************************************************************************)
VAR CONSTANT
	LOG_SW_OBJ_RM : UINT := 55022; (*Software object removed*)
	LOG_SW_OBJ_NEW : UINT := 55021; (*New software object*)
	LOG_SW_OBJ_CHG : UINT := 55020; (*Software object changed*)
	swListDatObjName : STRING[7] := 'swList'; (*Software list*)
	swListTempDataObjName : STRING[7] := 'swListT'; (*Temporary software list*)
END_VAR
